PROGRAM MAIN
VAR
 // Edge Detector
	inputValue: BOOL := FALSE;
myEDG_var  : EdgeDetector;
riesingEdge :BOOL;
fallingEdge :BOOL;
	
currentSafeState  : SafeState := 0;
	
END_VAR

CASE currentSafeState OF
	
0:


1:


2:


3:


4:

END_CASE

//Implement Edge Detector
myEDG_var();
myEDG_var.inputValue := inputValue;
// Outputs from Edge Detection
riesingEdge :=myEDG_var.riesingEdge;
fallingEdge :=myEDG_var.fallingEdge;

END_PROGRAM

(* stored: Version 1.1.0.1, ProductVersion 3.1.4022.12
   POU MAIN: Id {085c1498-bfec-42b5-9b30-2ef2e53ea97d}, SpecialFunc None *)
